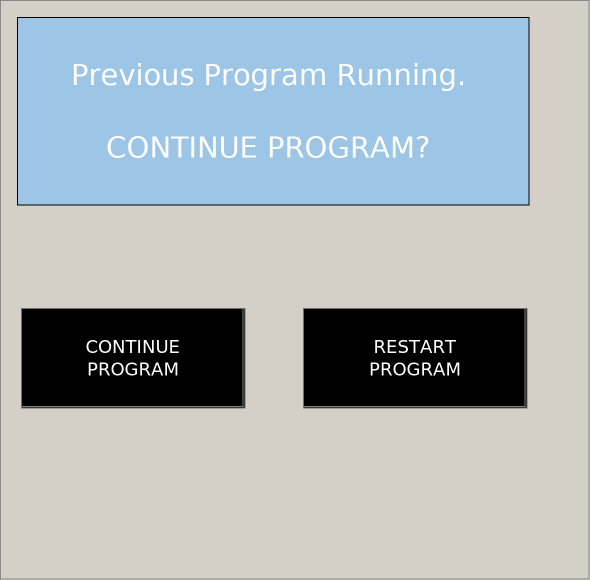
VISUALIZATION continueAutoScreen  // 590x580
    Textfield (17,17 512x188), "Previous Program Running. CONTINUE PROGRAM?"
    Button (21,308 224x100), "CONTINUE PROGRAM"
        toggle auto.bContinueProgBtn
    Button (303,308 224x100), "RESTART PROGRAM"
        toggle auto.bRestartProgBtn
END_VISUALIZATION

(* stored: Version 1.1.0.1, ProductVersion 3.1.4024.15
   Visu continueAutoScreen: Id {2c9b50d5-f7ef-4fb8-a031-a3847bd45c02} *)
